FUNCTION_BLOCK SERVO_RASPBERRY
  {SET_ATTRIBUTE(OpcUa, SERVICE)}
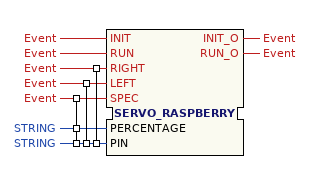
  EVENT_INPUT
    INIT;
    RUN;
    RIGHT WITH PIN;
    LEFT WITH PIN;
    SPEC WITH PERCENTAGE, PIN;
  END_EVENT
  EVENT_OUTPUT
    INIT_O;
    RUN_O;
  END_EVENT
  VAR_INPUT
    PERCENTAGE : STRING; {SET_ATTRIBUTE(OpcUa, Constant)}
    PIN : STRING; {SET_ATTRIBUTE(OpcUa, Constant)}
  END_VAR
END_FUNCTION_BLOCK
